FUNCTION_BLOCK MEASUREMENTS_TO_JSON_TIMESERIES
  {SET_ATTRIBUTE(OpcUa, POINT.ENDPOINT)}
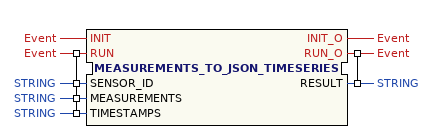
  EVENT_INPUT
    INIT;
    RUN WITH SENSOR_ID, MEASUREMENTS, TIMESTAMPS;
  END_EVENT
  EVENT_OUTPUT
    INIT_O;
    RUN_O WITH RESULT;
  END_EVENT
  VAR_INPUT
    SENSOR_ID : STRING; {SET_ATTRIBUTE(OpcUa, Constant.RUN)}
    MEASUREMENTS : STRING; {SET_ATTRIBUTE(OpcUa, Variable.RUN)}
    TIMESTAMPS : STRING; {SET_ATTRIBUTE(OpcUa, Variable.RUN)}
  END_VAR
  VAR_OUTPUT
    RESULT : STRING; {SET_ATTRIBUTE(OpcUa, Constant.RUN)}
  END_VAR
END_FUNCTION_BLOCK
